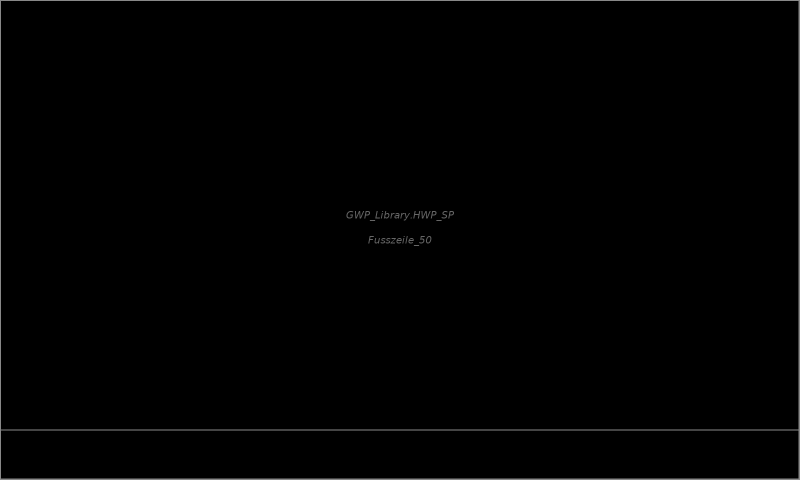
VISUALIZATION HWP_SP  // 800x480
    Frame (0,0 800x430)
        shows GWP_Library.HWP_SP(FB_HWP_SP := Main.HWP_SP_0, FB_KD := Main.KD_0)
    Frame (0,0 800x480)
        shows Fusszeile_50()
END_VISUALIZATION

(* stored: Version 1.1.0.1, ProductVersion 3.1.4022.6
   Visu HWP_SP: Id {55c6da92-574b-4ab3-b2c4-3826683ec2fb} *)
